FUNCTION_BLOCK FB_READ_HW
VAR_INPUT
END_VAR
VAR_OUTPUT
END_VAR
VAR
	ShuttleDebounce	: ARRAY[0..3] OF FB_DEBOUNCE;
END_VAR



ShuttleDebounce[0](SignalIn := IO.DI_Block_0[0], DebounceDelay := T#20MS);
ShuttleDebounce[1](SignalIn := IO.DI_Block_0[1], DebounceDelay := T#20MS);

// COMPONENT TESTING
SYS.Scale.ScaleIn.Status 			:= COM.COM1.StatusWord;
SYS.Scale.ScaleIn.InputLength 		:= COM.COM1.InputLength;
SYS.Scale.ScaleIn.Data 				:= COM.COM1.DataIn;

// MAIN INPUTS
PARAM.AUTO_MODE := IO.DI_Slice_0[0];
// PARAM.AUTO_MODE := TRUE;

// DEBINNER CELL (ROBOT)
SYS.RobotCell.RobotIN.RobotStatus 				:= ROBOT.Debinner.RobotStatus;
SYS.RobotCell.RobotIN.RobotAlarmStatus			:= ROBOT.Debinner.RobotAlarmStatus;
SYS.RobotCell.RobotIN.RobotAxisStatus 			:= ROBOT.Debinner.RobotAxisStatus;
SYS.RobotCell.RobotIN.RobotCycleStatus 			:= ROBOT.Debinner.RobotCycleStatus;
SYS.RobotCell.RobotIN.RobotJobSelectedStatus 	:= ROBOT.Debinner.RobotJobSelectedStatus;
SYS.RobotCell.RobotIN.RobotJobRunStatus 		:= ROBOT.Debinner.RobotJobRunStatus;
SYS.RobotCell.RobotIN.RobotJobCallStatus 		:= ROBOT.Debinner.RobotJobCallStatus;
SYS.RobotCell.RobotIN.RobotJobHoldStatus 		:= ROBOT.Debinner.RobotJobHoldStatus;
SYS.RobotCell.RobotIN.RobotJobHeldStatus 		:= ROBOT.Debinner.RobotJobHeldStatus;
SYS.RobotCell.RobotIN.RobotSystemStatus 		:= ROBOT.Debinner.RobotSystemStatus;
SYS.RobotCell.RobotIN.RobotUserInput			:= ROBOT.Debinner.RobotUserInput;
SYS.RobotCell.RobotIN.RobotAlarmCode1			:= ROBOT.Debinner.RobotAlarmCode1;
SYS.RobotCell.RobotIN.RobotAlarmCode2			:= ROBOT.Debinner.RobotAlarmCode2;
SYS.RobotCell.RobotIN.RobotErrorCode1			:= ROBOT.Debinner.RobotErrorCode1;
SYS.RobotCell.RobotIN.RobotErrorCode2			:= ROBOT.Debinner.RobotErrorCode2;
		
SYS.RobotCell.TraySense1						:= ShuttleDebounce[0].SignalOut;		
SYS.RobotCell.TraySense2						:= ShuttleDebounce[1].SignalOut;

SYS.RobotCell.RobotBuffer.OutFeedBufferSense	:= IO.DI_Block_0[2];
// SYS.RobotCell.TrayStuckDetection.TraySense		:= IO.DI_Block_0[3];			
SYS.RobotCell.TrayStuckDetection.TraySense1 	:= IO.DI_Block_0[3];				
SYS.RobotCell.TrayStuckDetection.TraySense2 	:= IO.DI_Block_0[4];			

SYS.RobotCell.AirPressureOK						:= IO.DI_Block_10[0];			// Need to map this to the hardware device
// SYS.RobotCell.AirPressureOK						:= TRUE;					// Air pressure error override (until switch is mechanically installed)

// PACK STATION INFEED CONVEYOR (VFD)
SYS.PackStation.InFeedConvIn.StatusWord 	:= MOTORS.PackInFeedConv.StatusWord;
SYS.PackStation.InFeedConvIn.ErrorCode 		:= MOTORS.PackInFeedConv.ErrorCode;
SYS.PackStation.InFeedConvIn.ActualVelocity := MOTORS.PackInFeedConv.ActualVelocity;

// PACK STATION OUTFEED CONVEYOR (VFD)
SYS.PackStation.OutFeedConvIn.StatusWord 		:= MOTORS.PackOutFeedConv.StatusWord;
SYS.PackStation.OutFeedConvIn.ErrorCode 		:= MOTORS.PackOutFeedConv.ErrorCode;
SYS.PackStation.OutFeedConvIn.ActualVelocity 	:= MOTORS.PackOutFeedConv.ActualVelocity;

// PACK STATION ROTARY ACCUMULATOR (VFD)
SYS.PackStation.RotaryAccumulatorIn.StatusWord		:= MOTORS.RotaryAccumulator.StatusWord;
SYS.PackStation.RotaryAccumulatorIn.ErrorCode		:= MOTORS.RotaryAccumulator.ErrorCode;
SYS.PackStation.RotaryAccumulatorIn.ActualVelocity	:= MOTORS.RotaryAccumulator.ActualVelocity;

// FRESH FRUIT DEBIN CONVEYOR (VFD)
SYS.FreshFruit.DebinConvIN.StatusWord 		:= MOTORS.DebinConv.StatusWord;
SYS.FreshFruit.DebinConvIN.ErrorCode 		:= MOTORS.DebinConv.ErrorCode;
SYS.FreshFruit.DebinConvIN.ActualVelocity 	:= MOTORS.DebinConv.ActualVelocity;

// FRESH FRUIT SORT CONVEYOR (VFD)
SYS.FreshFruit.SortConvIN.StatusWord 		:= MOTORS.SortConv.StatusWord;
SYS.FreshFruit.SortConvIN.ErrorCode 		:= MOTORS.SortConv.ErrorCode;
SYS.FreshFruit.SortConvIN.ActualVelocity 	:= MOTORS.SortConv.ActualVelocity;

// FRESH FRUIT LANING CONVEYOR (VFD)
SYS.FreshFruit.LaneConvIN.StatusWord 		:= MOTORS.LaneConv.StatusWord;
SYS.FreshFruit.LaneConvIN.ErrorCode 		:= MOTORS.LaneConv.ErrorCode;
SYS.FreshFruit.LaneConvIN.ActualVelocity 	:= MOTORS.LaneConv.ActualVelocity;

// ROBOT CELL INFEED CONVEYOR (VFD)
SYS.RobotCell.InFeedConvIN.StatusWord 			:= MOTORS.RobotInFeedConv.StatusWord;
SYS.RobotCell.InFeedConvIN.OperationModeDisplay := MOTORS.RobotInFeedConv.OperationModeDisplay;
SYS.RobotCell.InFeedConvIN.ActualVelocity 		:= MOTORS.RobotInFeedConv.ActualVelocity;

// ROBOT CELL OUTFEED CONVEYOR (VFD)
SYS.RobotCell.OutFeedConvIN.StatusWord 				:= MOTORS.RobotOutFeedConv.StatusWord;
SYS.RobotCell.OutFeedConvIN.OperationModeDisplay 	:= MOTORS.RobotOutFeedConv.OperationModeDisplay;
SYS.RobotCell.OutFeedConvIN.ActualVelocity 			:= MOTORS.RobotOutFeedConv.ActualVelocity;

// FILL STATION INFEED CONVEYOR (VFD)
SYS.FillStation.InFeedConvIN.StatusWord 			:= MOTORS.FillInFeedConv.StatusWord;
SYS.FillStation.InFeedConvIN.OperationModeDisplay 	:= MOTORS.FillInFeedConv.OperationModeDisplay;
SYS.FillStation.InFeedConvIN.ActualVelocity 		:= MOTORS.FillInFeedConv.ActualVelocity;
SYS.FillStation.InFeedConvIN.MotorCurrent			:= MOTORS.FillInFeedConv.MotorCurrent;
SYS.FillStation.InFeedConvIN.MotorPowerEff			:= MOTORS.FillInFeedConv.MotorPowerEff;

// DENESTER 0 (IO)
SYS.Denester[0].VacSense1 := IO.DI_Block_4[0];
SYS.Denester[0].VacSense2 := IO.DI_Block_4[1];
SYS.Denester[0].ExtendEOT := IO.DI_Block_4[2];

// DENESTER 1 (IO)
SYS.Denester[1].VacSense1 := IO.DI_Block_3[0];
SYS.Denester[1].VacSense2 := IO.DI_Block_3[1];
SYS.Denester[1].ExtendEOT := IO.DI_Block_3[2];

// DENESTER 2 (IO)
SYS.Denester[2].VacSense1 := IO.DI_Block_2[0];
SYS.Denester[2].VacSense2 := IO.DI_Block_2[1];
SYS.Denester[2].ExtendEOT := IO.DI_Block_2[2];

// DENESTER 3 (IO)
SYS.Denester[3].VacSense1 := IO.DI_Block_1[0];
SYS.Denester[3].VacSense2 := IO.DI_Block_1[1];
SYS.Denester[3].ExtendEOT := IO.DI_Block_1[2];

// DENESTER BUFFER SENSORS / FILL STATION JAM SENSORS (IO)
// SYS.Denester[0].ClamBuffer.BufferSense1 := IO.DI_Block_8[0];
// SYS.Denester[0].Clambuffer.BufferSense2 := IO.DI_Block_8[1];
SYS.Denester[0].ClamBufferNew.BufferSense1 := IO.DI_Block_8[0];
SYS.Denester[0].ClambufferNew.BufferSense2 := IO.DI_Block_8[1];
// SYS.Denester[1].ClamBuffer.BufferSense1 := IO.DI_Block_8[2];
// SYS.Denester[1].Clambuffer.BufferSense2 := IO.DI_Block_8[3];
SYS.Denester[1].ClamBufferNew.BufferSense1 := IO.DI_Block_8[2];
SYS.Denester[1].ClambufferNew.BufferSense2 := IO.DI_Block_8[3];
// SYS.Denester[2].ClamBuffer.BufferSense1 := IO.DI_Block_8[4];
// SYS.Denester[2].Clambuffer.BufferSense2 := IO.DI_Block_8[5];
SYS.Denester[2].ClamBufferNew.BufferSense1 := IO.DI_Block_8[13];			// Old port #4, new port #13
SYS.Denester[2].ClambufferNew.BufferSense2 := IO.DI_Block_8[5];
// SYS.Denester[3].ClamBuffer.BufferSense1 := IO.DI_Block_8[6];
// SYS.Denester[3].Clambuffer.BufferSense2 := IO.DI_Block_8[7];
SYS.Denester[3].ClamBufferNew.BufferSense1 := IO.DI_Block_8[6];
SYS.Denester[3].ClambufferNew.BufferSense2 := IO.DI_Block_8[7];

SYS.FillStation.FillBuffer[0].BufferSense := IO.DI_Block_8[8];	// Originally DI_Block_8[8]
SYS.FillStation.FillBuffer[1].BufferSense := IO.DI_Block_8[10];	// Originally DI_Block_8[10]
SYS.FillStation.FillBuffer[2].BufferSense := IO.DI_Block_8[12];	// Originally DI_Block_8[12]
SYS.FillStation.FillBuffer[3].BufferSense := IO.DI_Block_8[14];	// Originally DI_Block_8[14]

// JUICE COLLECTION CONVEYOR (VFD)
SYS.Juice.CollectConvIN.StatusWord 				:= MOTORS.JuiceCollectConv.StatusWord;
SYS.Juice.CollectConvIN.OperationModeDisplay 	:= MOTORS.JuiceCollectConv.OperationModeDisplay;
SYS.Juice.CollectConvIN.ActualVelocity 			:= MOTORS.JuiceCollectConv.ActualVelocity;

// JUICE DISCHARGE CONVEYOR (VFD)
SYS.Juice.DischargeConvIN.StatusWord 			:= MOTORS.JuiceDischargeConv.StatusWord;
SYS.Juice.DischargeConvIN.OperationModeDisplay 	:= MOTORS.JuiceDischargeConv.OperationModeDisplay;
SYS.Juice.DischargeConvIN.ActualVelocity 		:= MOTORS.JuiceDischargeConv.ActualVelocity;

// JUICE INFEED CONVEYOR (VFD)
SYS.Juice.InFeedConvIN.StatusWord 				:= MOTORS.JuiceInFeedConv.StatusWord;
SYS.Juice.InFeedConvIN.OperationModeDisplay 	:= MOTORS.JuiceInFeedConv.OperationModeDisplay;
SYS.Juice.InFeedConvIN.ActualVelocity 			:= MOTORS.JuiceInFeedConv.ActualVelocity;

// JUICE OUTFEED CONVEYOR (VFD)
SYS.Juice.OutFeedConvIN.StatusWord 				:= MOTORS.JuiceOutFeedConv.StatusWord;
SYS.Juice.OutFeedConvIN.OperationModeDisplay 	:= MOTORS.JuiceOutFeedConv.OperationModeDisplay;
SYS.Juice.OutFeedConvIN.ActualVelocity 			:= MOTORS.JuiceOutFeedConv.ActualVelocity;

// FILL STATION MOTOR 0 (PD4)
SYS.FillStation.PD4IN[0].StatusWord 				:= MOTORS.FillStationMotor[3].StatusWord;
SYS.FillStation.PD4IN[0].OperationModeDisplay 		:= MOTORS.FillStationMotor[3].OperationModeDisplay;
SYS.FillStation.PD4IN[0].ActualPosition 			:= MOTORS.FillStationMotor[3].ActualPosition;

// FILL STATION MOTOR 1 (PD4)
SYS.FillStation.PD4IN[1].StatusWord 				:= MOTORS.FillStationMotor[2].StatusWord;
SYS.FillStation.PD4IN[1].OperationModeDisplay 		:= MOTORS.FillStationMotor[2].OperationModeDisplay;
SYS.FillStation.PD4IN[1].ActualPosition 			:= MOTORS.FillStationMotor[2].ActualPosition;

// FILL STATION MOTOR 2 (PD4)
SYS.FillStation.PD4IN[2].StatusWord 				:= MOTORS.FillStationMotor[1].StatusWord;
SYS.FillStation.PD4IN[2].OperationModeDisplay 		:= MOTORS.FillStationMotor[1].OperationModeDisplay;
SYS.FillStation.PD4IN[2].ActualPosition 			:= MOTORS.FillStationMotor[1].ActualPosition;

// FILL STATION MOTOR 3 (PD4)
SYS.FillStation.PD4IN[3].StatusWord 				:= MOTORS.FillStationMotor[0].StatusWord;
SYS.FillStation.PD4IN[3].OperationModeDisplay 		:= MOTORS.FillStationMotor[0].OperationModeDisplay;
SYS.FillStation.PD4IN[3].ActualPosition 			:= MOTORS.FillStationMotor[0].ActualPosition;

// FILL STATION SENSOR ARRAYS
SYS.FillStation.SenseArray[0].SenseArray[0] := IO.DI_Block_6[0];
SYS.FillStation.SenseArray[0].SenseArray[1] := IO.DI_Block_6[1];
SYS.FillStation.SenseArray[0].SenseArray[2] := IO.DI_Block_6[2];
SYS.FillStation.SenseArray[0].SenseArray[3] := IO.DI_Block_6[3];
SYS.FillStation.SenseArray[0].SenseArray[4] := IO.DI_Block_6[4];
SYS.FillStation.SenseArray[0].SenseArray[5] := IO.DI_Block_6[5];
SYS.FillStation.SenseArray[0].SenseArray[6] := IO.DI_Block_6[6];
SYS.FillStation.SenseArray[0].SenseArray[7] := IO.DI_Block_6[7];

SYS.FillStation.SenseArray[1].SenseArray[0] := IO.DI_Block_6[8];
SYS.FillStation.SenseArray[1].SenseArray[1] := IO.DI_Block_6[9];
SYS.FillStation.SenseArray[1].SenseArray[2] := IO.DI_Block_6[10];
SYS.FillStation.SenseArray[1].SenseArray[3] := IO.DI_Block_6[11];
SYS.FillStation.SenseArray[1].SenseArray[4] := IO.DI_Block_6[12];
SYS.FillStation.SenseArray[1].SenseArray[5] := IO.DI_Block_6[13];
SYS.FillStation.SenseArray[1].SenseArray[6] := IO.DI_Block_6[14];
SYS.FillStation.SenseArray[1].SenseArray[7] := IO.DI_Block_6[15];

SYS.FillStation.SenseArray[2].SenseArray[0] := IO.DI_Block_7[0];
SYS.FillStation.SenseArray[2].SenseArray[1] := IO.DI_Block_7[1];
SYS.FillStation.SenseArray[2].SenseArray[2] := IO.DI_Block_7[2];
SYS.FillStation.SenseArray[2].SenseArray[3] := IO.DI_Block_7[3];
SYS.FillStation.SenseArray[2].SenseArray[4] := IO.DI_Block_7[4];
SYS.FillStation.SenseArray[2].SenseArray[5] := IO.DI_Block_7[5];
SYS.FillStation.SenseArray[2].SenseArray[6] := IO.DI_Block_7[6];
SYS.FillStation.SenseArray[2].SenseArray[7] := IO.DI_Block_7[7];

SYS.FillStation.SenseArray[3].SenseArray[0] := IO.DI_Block_7[8];
SYS.FillStation.SenseArray[3].SenseArray[1] := IO.DI_Block_7[9];
SYS.FillStation.SenseArray[3].SenseArray[2] := IO.DI_Block_7[10];
SYS.FillStation.SenseArray[3].SenseArray[3] := IO.DI_Block_7[11];
SYS.FillStation.SenseArray[3].SenseArray[4] := IO.DI_Block_7[12];
SYS.FillStation.SenseArray[3].SenseArray[5] := IO.DI_Block_7[13];
SYS.FillStation.SenseArray[3].SenseArray[6] := IO.DI_Block_7[14];
SYS.FillStation.SenseArray[3].SenseArray[7] := IO.DI_Block_7[15];

// 	PACK STATION BUFFER SENSOR INPUTS
SYS.PackStation.PackBufferSense[0] := IO.DI_Block_9[0];
SYS.PackStation.PackBufferSense[1] := IO.DI_Block_9[1];
SYS.PackStation.PackBufferSense[2] := IO.DI_Block_9[2];
SYS.PackStation.PackBufferSense[3] := IO.DI_Block_9[3];

// JUICE INPUTS
SYS.Juice.JuiceBox.JuiceBoxIn := IO.DI_Block_5[0];

// JUICE SERIAL COM (SCALE)
SYS.Juice.JuiceScaleIn.Status 		:= COM.JuiceScale.StatusWord;
SYS.Juice.JuiceScaleIn.InputLength 	:= COM.JuiceScale.InputLength;
SYS.Juice.JuiceScaleIn.Data 		:= COM.JuiceScale.DataIn;

// PACK STATION SERIAL COM 0 (SCALE)
SYS.PackStation.ScaleIn[0].Status			:= COM.PackScale[0].StatusWord;
SYS.PackStation.ScaleIn[0].InputLength 		:= COM.PackScale[0].InputLength;
SYS.PackStation.ScaleIn[0].Data 			:= COM.PackScale[0].DataIn;

// PACK STATION SERIAL COM 1 (SCALE)
SYS.PackStation.ScaleIn[1].Status			:= COM.PackScale[1].StatusWord;
SYS.PackStation.ScaleIn[1].InputLength 		:= COM.PackScale[1].InputLength;
SYS.PackStation.ScaleIn[1].Data 			:= COM.PackScale[1].DataIn;

// PACK STATION SERIAL COM 2 (SCALE)
SYS.PackStation.ScaleIn[2].Status			:= COM.PackScale[2].StatusWord;
SYS.PackStation.ScaleIn[2].InputLength 		:= COM.PackScale[2].InputLength;
SYS.PackStation.ScaleIn[2].Data 			:= COM.PackScale[2].DataIn;

// PACK STATION SERIAL COM 3 (SCALE)
SYS.PackStation.ScaleIn[3].Status			:= COM.PackScale[3].StatusWord;
SYS.PackStation.ScaleIn[3].InputLength 		:= COM.PackScale[3].InputLength;
SYS.PackStation.ScaleIn[3].Data 			:= COM.PackScale[3].DataIn;

// PACK STATION SERIAL COM 4 (SCALE)
SYS.PackStation.ScaleIn[4].Status			:= COM.PackScale[4].StatusWord;
SYS.PackStation.ScaleIn[4].InputLength 		:= COM.PackScale[4].InputLength;
SYS.PackStation.ScaleIn[4].Data 			:= COM.PackScale[4].DataIn;

// PACK STATION SERIAL COM 5 (SCALE)
SYS.PackStation.ScaleIn[5].Status			:= COM.PackScale[5].StatusWord;
SYS.PackStation.ScaleIn[5].InputLength 		:= COM.PackScale[5].InputLength;
SYS.PackStation.ScaleIn[5].Data 			:= COM.PackScale[5].DataIn;

// PACK STATION SERIAL COM 6 (SCALE)
SYS.PackStation.ScaleIn[6].Status			:= COM.PackScale[6].StatusWord;
SYS.PackStation.ScaleIn[6].InputLength 		:= COM.PackScale[6].InputLength;
SYS.PackStation.ScaleIn[6].Data 			:= COM.PackScale[6].DataIn;

// PACK STATION SERIAL COM 7 (SCALE)
SYS.PackStation.ScaleIn[7].Status			:= COM.PackScale[7].StatusWord;
SYS.PackStation.ScaleIn[7].InputLength 		:= COM.PackScale[7].InputLength;
SYS.PackStation.ScaleIn[7].Data 			:= COM.PackScale[7].DataIn;

// PACK STATION SERIAL COM 8 (SCALE)
SYS.PackStation.ScaleIn[8].Status			:= COM.PackScale[8].StatusWord;
SYS.PackStation.ScaleIn[8].InputLength 		:= COM.PackScale[8].InputLength;
SYS.PackStation.ScaleIn[8].Data 			:= COM.PackScale[8].DataIn;

// PACK STATION SERIAL COM 9 (SCALE)
SYS.PackStation.ScaleIn[9].Status			:= COM.PackScale[9].StatusWord;
SYS.PackStation.ScaleIn[9].InputLength 		:= COM.PackScale[9].InputLength;
SYS.PackStation.ScaleIn[9].Data 			:= COM.PackScale[9].DataIn;

// PACK STATION SERIAL COM 10 (SCALE)
SYS.PackStation.ScaleIn[10].Status			:= COM.PackScale[10].StatusWord;
SYS.PackStation.ScaleIn[10].InputLength 	:= COM.PackScale[10].InputLength;
SYS.PackStation.ScaleIn[10].Data 			:= COM.PackScale[10].DataIn;

// PACK STATION SERIAL COM 11 (SCALE)
SYS.PackStation.ScaleIn[11].Status			:= COM.PackScale[11].StatusWord;
SYS.PackStation.ScaleIn[11].InputLength 	:= COM.PackScale[11].InputLength;
SYS.PackStation.ScaleIn[11].Data 			:= COM.PackScale[11].DataIn;

END_FUNCTION_BLOCK

(* stored: Version 1.1.0.1, ProductVersion 3.1.4024.12
   POU FB_READ_HW: Id {38d0a033-22ac-41e8-ba5b-56b320f7ade6}, SpecialFunc None *)
